INTERFACE I_TracePublisher

METHOD Subscribe
VAR_INPUT
	Logger : I_TraceLogger;
END_VAR

VAR
	i : UDINT;
END_VAR
END_METHOD

METHOD Unsubscribe
VAR_INPUT
	Logger : I_TraceLogger;
END_VAR

VAR
	i : UDINT;
END_VAR
END_METHOD

END_INTERFACE

(* stored: Version 1.1.0.1
   Itf I_TracePublisher: Id {527d72c4-d8e1-4604-87b2-42428273b381}
   Method Subscribe: Id {893f19fc-463e-439e-a8b0-79ed859ec4ed}
   Method Unsubscribe: Id {31120338-b3a2-428f-b659-bf8777f2bc79} *)
